# EPICS alarm handler configuration: mps_database/bareTest/alarms/areas/mpln_gunb_mp02.alhConfig
GROUP NULL MPLN:GUNB:MP02:1
$ALIAS MPS Link Node 49
$GUIDANCE
LTUH MPS
   Group Name: MPLN:GUNB:MP02:1
   Summary PV:  MPLN:GUNB:MP02:1:STATSUMY
$END
CHANNEL  MPLN:GUNB:MP02:1    MPLN:GUNB:MP02:1:MPS_EN_RBV		-----
CHANNEL  MPLN:GUNB:MP02:1    MPLN:GUNB:MP02:1:LC1_MODE_RBV		-----
